// TwinCAT 3 PLC project TempModel
// ProgramVersion: 3.1.4026.20
// libraries:
//   Tc2_Standard, * (Beckhoff Automation GmbH)
//   Tc2_System, * (Beckhoff Automation GmbH)
//   Tc3_Module, * (Beckhoff Automation GmbH)
// project tree:
//   GVLs/ GVL_1654353297.TcGVL
//   / PlcTask.TcTTO
//   POUs/ MAIN.TcPOU, Temp_Model0.TcPOU
// real-time tasks:
//   TASK PlcTask: cycle T#10ms, priority 21, ADS port 350
//   TASK PlcTask1: cycle T#10ms, priority 22, ADS port 351
//   TASK PlcTask2: cycle T#10ms, priority 20, ADS port 352
// motion (NC):
//   TASK NC-Task 1 SAF: cycle T#2ms, priority 4, ADS port 501
//   TASK NC-Task 1 SVB: cycle T#10ms, priority 8, ADS port 511
//   AXIS BandAchse (id 1)
//     Dynamic: AccelerationMaximum=200, DecelerationMaximum=200, Acceleration=150, Deceleration=150
//     Velo: SlowManual=20, FastManual=50, Maximum=50
//     OtherSettings: AllowMotionCmdToSlave=true
//     encoder EncType=16
//       EncPara: MaxCount=#x0000ffff
//     drive DrvType=13
//       Analog: VeloReferenz=60, TorqueSetpointScale=10, ScaleFactorActTorque=0.1
//       TimeComp: TaskDelayCycles=1
//     controller CtrType=1
//       CtrPara: PriorControlFactor=1
//         Observer: BandWidth=20
// variable links:
//   LF_System_PLC/LF_System_PLC Instance <-> NC-Task 1 SAF/Axes/BandAchse
//     PlcTask Inputs/MAIN.fIN_CnvPos <-> Outputs/ToPlc/ActPos
//   LF_System_PLC/LF_System_PLC Instance <-> PLC/PLC Instance
//     PlcTask Inputs/MAIN.bIn_LedGreen <-> PlcTask Outputs/IFC_HW.bAmpelGrun
//     PlcTask Inputs/MAIN.bIn_LedRot <-> PlcTask Outputs/IFC_HW.bAmpelRot
//     PlcTask Inputs/MAIN.bIn_LedYellow <-> PlcTask Outputs/IFC_HW.bAmpelGelb
//     PlcTask Inputs/MAIN.bIn_Schleuse1_L1 <-> PlcTask Outputs/IFC_HW.bR1AKT1
//     PlcTask Inputs/MAIN.bIn_Schleuse1_L2 <-> PlcTask Outputs/IFC_HW.bR2AKT1
//     PlcTask Inputs/MAIN.bIn_Schleuse2_L1 <-> PlcTask Outputs/IFC_HW.bR1AKT2
//     PlcTask Inputs/MAIN.bIn_Schleuse2_L2 <-> PlcTask Outputs/IFC_HW.bR2AKT2
//     PlcTask Outputs/MAIN.bEnable <-> PlcTask Inputs/IFC_HW.bEnable
//     PlcTask Outputs/MAIN.bExecute <-> PlcTask Inputs/IFC_HW.bExecute
//     PlcTask Outputs/MAIN.bOut_VereinzelungNS1 <-> PlcTask Inputs/IFC_HW.bEinzelSens3
//     PlcTask Outputs/MAIN.bOut_VereinzelungNS2 <-> PlcTask Inputs/IFC_HW.bEinzelSens2
//     PlcTask Outputs/MAIN.bOut_VereinzelungNS3 <-> PlcTask Inputs/IFC_HW.bEinzelSens1
//   PLC/PLC Instance <-> NC-Task 1 SAF/Axes/BandAchse
//     PlcTask Inputs/IFC_HW.ax_BandMotor.NcToPlc <-> Outputs/ToPlc
//     PlcTask Outputs/IFC_HW.ax_BandMotor.PlcToNc <-> Inputs/FromPlc

CONFIGURATION TempModel
    RESOURCE PLC ON TwinCAT3
        TASK PlcTask(INTERVAL := T#10ms, PRIORITY := 21);
        PROGRAM MAIN WITH PlcTask : MAIN;
    END_RESOURCE
END_CONFIGURATION

// ---- GVLs/GVL_1654353297.TcGVL
VAR_GLOBAL CONSTANT
	SS_INITIALIZE: SINT := 0;
	SS_STEP: SINT := 1;
END_VAR

// ---- POUs/MAIN.TcPOU
PROGRAM MAIN
VAR
iVolt 		AT%I* : UINT;
iTempSens1 	AT%Q* : UINT;
iTempSens2 	AT%Q* : UINT;
fbTempModel : Temp_Model0;
END_VAR


fbTempModel(ssMethodType:= , iVolt_U:= iVolt , iTemp1_Y=> iTempSens1 , iTemp2_Y=> iTempSens2 );
fbTempModel.ssMethodType := 1;

END_PROGRAM

// ---- POUs/Temp_Model0.TcPOU
FUNCTION_BLOCK Temp_Model0
VAR_INPUT
	ssMethodType: SINT := 0;
	iVolt_U: UINT;
END_VAR
VAR_OUTPUT
	iTemp1_Y: UINT;
	iTemp2_Y: UINT;
END_VAR
VAR
	rtb_Gain1: LREAL;
	rtb_Add1: LREAL;
	i: DINT;
	rtb_DiscreteTransferFcn: LREAL;
	DiscreteTransferFcn_states: LREAL;
	b_counter: DINT;
	counter_b: DINT;
	Delay_DSTATE: ARRAY[0..2279] OF LREAL;
END_VAR



CASE ssMethodType OF
    SS_INITIALIZE: 
        (* SystemInitialize for Atomic SubSystem: '<Root>/Temp_Model' *)
        (* InitializeConditions for Sin: '<S1>/Sine Wave' *)
        b_counter := 0;
        (* End of SystemInitialize for SubSystem: '<Root>/Temp_Model' *)
        (* SystemInitialize for Atomic SubSystem: '<Root>/Temp_Model' *)
        (* InitializeConditions for Delay: '<S1>/Delay' *)

        FOR i := 0 TO 2279 DO 
            Delay_DSTATE[i] := 0.0;
        END_FOR;

        (* End of InitializeConditions for Delay: '<S1>/Delay' *)
        

        (* InitializeConditions for Sin: '<S1>/Sine Wave1' *)
        counter_b := 0;
        (* InitializeConditions for DiscreteTransferFcn: '<S1>/Discrete Transfer Fcn' *)
        DiscreteTransferFcn_states := 0.0;
        (* End of SystemInitialize for SubSystem: '<Root>/Temp_Model' *)
    SS_STEP: 
        (* Outputs for Atomic SubSystem: '<Root>/Temp_Model' *)
        (* Sum: '<S1>/Add1' incorporates:
         *  Constant: '<S1>/T_umg1'
         *  Delay: '<S1>/Delay'
         *  Sin: '<S1>/Sine Wave'
         *  Sum: '<S1>/Sum5' *)
        rtb_Add1 := (SIN(((DINT_TO_LREAL(b_counter) * 2.0) * 3.1415926535897931) / 100.0) * 0.3) + (Delay_DSTATE[0] + 25.0);
        (* Sum: '<S1>/Add' incorporates:
         *  Constant: '<S1>/T_umg1'
         *  Delay: '<S1>/Delay'
         *  Sin: '<S1>/Sine Wave1'
         *  Sum: '<S1>/Sum5' *)
        rtb_Gain1 := (SIN(((DINT_TO_LREAL(counter_b) * 2.0) * 3.1415926535897931) / 100.0 + 1.57) * 0.2) + (Delay_DSTATE[0] + 25.0);
        (* DiscreteTransferFcn: '<S1>/Discrete Transfer Fcn' incorporates:
         *  DataTypeConversion: '<S1>/Data Type Conversion'
         *  Gain: '<S1>/D//A-Wandler EL4002' *)
        rtb_DiscreteTransferFcn := (0.00015259254737998596 * UINT_TO_LREAL(iVolt_U)) - (-0.99996221812467 * DiscreteTransferFcn_states);
        (* Update for Sin: '<S1>/Sine Wave' *)
        b_counter := b_counter + 1;

        IF b_counter = 1000 THEN 
            b_counter := 0;
        END_IF;

        (* End of Update for Sin: '<S1>/Sine Wave' *)
        

        (* Update for Delay: '<S1>/Delay' incorporates:
         *  DiscreteTransferFcn: '<S1>/Discrete Transfer Fcn' *)

        FOR i := 0 TO 2278 DO 
            Delay_DSTATE[i] := Delay_DSTATE[i + 1];
        END_FOR;

        Delay_DSTATE[2279] := (0.000408383380313031 * rtb_DiscreteTransferFcn) + (0.000769303707329493 * DiscreteTransferFcn_states);
        (* End of Update for Delay: '<S1>/Delay' *)
        

        (* Update for Sin: '<S1>/Sine Wave1' *)
        counter_b := counter_b + 1;

        IF counter_b = 1000 THEN 
            counter_b := 0;
        END_IF;

        (* End of Update for Sin: '<S1>/Sine Wave1' *)
        

        (* Update for DiscreteTransferFcn: '<S1>/Discrete Transfer Fcn' *)
        DiscreteTransferFcn_states := rtb_DiscreteTransferFcn;
        (* Outport: '<Root>/iTemp1_Y' incorporates:
         *  DataTypeConversion: '<S1>/Data Type Conversion1'
         *  Gain: '<S1>/Gain' *)
        iTemp1_Y := DINT_TO_UINT(TRUNC(100.0 * rtb_Add1));
        (* Outport: '<Root>/iTemp2_Y' incorporates:
         *  DataTypeConversion: '<S1>/Data Type Conversion2'
         *  Gain: '<S1>/Gain1' *)
        iTemp2_Y := DINT_TO_UINT(TRUNC(100.0 * rtb_Gain1));
        (* End of Outputs for SubSystem: '<Root>/Temp_Model' *)
END_CASE;

END_FUNCTION_BLOCK
